(* PLC project First Test, Almighty ZRT11 TEST ST PLC 0.1.23.456 *)
(* stored: creationDateTime 1990-01-01T12:00:00, modificationDateTime 2016-04-10T17:37:00 *)

PROGRAM Ontarto
  VAR
    input1 AT %IX0.0 : BOOL;
    stop AT %MX0.0 : BOOL;
    output AT %QX0.0 : BOOL;
  END_VAR

									
									output := input1 OR output;
									IF
									 stop THEN output := FALSE;
									END_IF;
									
								
END_PROGRAM

PROGRAM StateInExample
  VAR
    input AT %IX0.0 : BOOL;
    output AT %QX0.0 : BOOL;
  END_VAR

									
									output := input;
									
								
END_PROGRAM

CONFIGURATION Application
  RESOURCE Application ON PLC
    TASK ExampleTask(INTERVAL := T#20ms, PRIORITY := 1);
    PROGRAM Ontarto WITH ExampleTask : Ontarto;
  END_RESOURCE
END_CONFIGURATION
